FUNCTION_BLOCK FB_S
VAR_INPUT

END_VAR
VAR_OUTPUT
	bValve				:BOOL;
END_VAR
VAR
	bValveOpen			:BOOL;	//SB Testing TRUE
	bValveClosed		:BOOL;	//SK
	bPrevOpen			:BOOL;
	bPrevClosed			:BOOL;	

	//on/off buttons or every 90 sec for 30sec if tank not empty
	nState				:UDINT := 0; //0: Default, 20: Autorun 40: Manual
	myTimer				:TON;
	tCurrentTime		:TIME;
	bTemp				:BOOL;
END_VAR

CASE nState OF
	0: //Scanning for Errors
		IF GVL.bHeatRelay OR GVL.bTankEmpty THEN
			//Error log
			bValve := FALSE;
			nState := 0;		//Stay in standby state 0
		ELSE
			nState := 20;
		END_IF
	20:	//Auto Closed
		IF GVL.bManualValve THEN
			nState := 60;
		END_IF;
		tCurrentTime := GVL.tValveOffTimer;
		bValve := FALSE;
		IF myTimer.Q THEN
			nState := 40;	
			myTimer(IN := FALSE);
		END_IF
	40: //Auto Open
		IF GVL.bManualValve THEN
			nState := 60;
		END_IF;
		tCurrentTime := GVL.tValveOnTimer;
		bValve := TRUE;
		IF myTimer.Q THEN
			nState := 0;
			myTimer(IN := FALSE);
		END_IF
		
	60:
		IF (bValveOpen AND NOT bPrevOpen) THEN
			bValveClosed:=FALSE;
			bValve := TRUE;
		ELSIF (BValveClosed AND NOT bPrevClosed) THEN
			BValveOpen:=FALSE;
			bValve := FALSE;		
		END_IF
		
		bPrevOpen := bValveOpen;
		bPrevClosed := bValveClosed;		
		
		IF NOT GVL.bManualValve THEN
			nState := 0;
		ELSE
			nState := 60;
		END_IF
END_CASE

myTimer(IN:=TRUE, PT:=tCurrentTime);
myTimer(IN:=TRUE, PT:=tCurrentTime);

END_FUNCTION_BLOCK

(* stored: Version 1.1.0.1, ProductVersion 3.1.4024.12
   POU FB_S: Id {bc0c4985-e852-4aab-b4a9-dbc3ff35f74d}, SpecialFunc None *)
